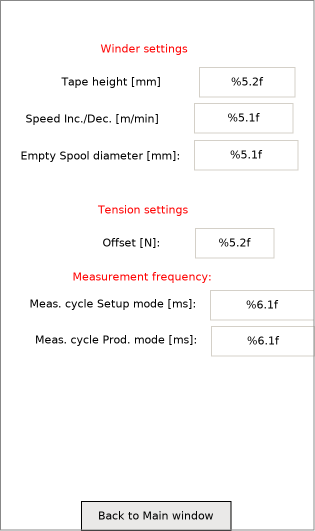
VISUALIZATION GeneralSettings  // 315x531
    Rectangle (81,501 150x30), "Back to Main window"
        OnMouseClick: change screen: MainWindow
    Textfield (199,67 96x30), "%5.2f", text variable: GVL_Parameter.TapeHeight
    Label (42,67 122x30), "Tape height [mm]"
    Label (69,34 150x30), "Winder settings"
    Textfield (194,103 99x30), "%5.1f", tooltip "Speed increment and decrement applied using the control pad.", text variable: GVL_Parameter.SpeedChange
        OnMouseClick: write GVL_Parameter.SpeedChange via VisuDialogs.Numpad
    Label (16,104 146x30), "Speed Inc./Dec. [m/min]"
    Textfield (195,228 79x30), "%5.2f"
    Label (41,228 122x30), "Offset [N]:"
    Label (68,195 150x30), "Tension settings"
    Textfield (194,140 104x30), "%5.1f", tooltip "Required to calculate speed reference value for winder motor.", text variable: GVL_Parameter.EmptySpoolDiameter
        OnMouseClick: write GVL_Parameter.EmptySpoolDiameter via VisuDialogs.Numpad, min 10, max 1000
    Label (16,141 167x30), "Empty Spool diameter [mm]:"
    Textfield (210,290 104x30), "%6.1f", tooltip "Defines how often measurements will be taken and written to a file. Lower values will increase the file size.", text variable: GVL_Parameter.tMeas_SetupMode
        OnMouseClick: write GVL_Parameter.tMeas_SetupMode via VisuDialogs.Numpad, min 10, max 100000, format 1000
    Label (14,289 185x30), "Meas. cycle Setup mode [ms]:"
    Textfield (211,326 104x30), "%6.1f", tooltip "Defines how often measurements will be taken and written to a file. Lower values will increase the file size.", text variable: GVL_Parameter.tMeas_ProductionMode
        OnMouseClick: write GVL_Parameter.tMeas_ProductionMode via Edit, min 10, max 100000, format 1000
    Label (15,325 185x30), "Meas. cycle Prod. mode [ms]:"
    Label (67,262 150x30), "Measurement frequency:"
END_VISUALIZATION

(* stored: Version 1.1.0.1
   Visu GeneralSettings: Id {85b79585-70bb-49d3-88bb-2b6392c9bd91} *)
